FUNCTION_BLOCK Valvula_Saida_Digital_HMI (* Service Interface Function Block Type *)
  (* Standard: 61499-2 *)
  (* Version 0.0, 1/26/2026, Schneider Electric, template *)
  PACKAGE Hidryco.HidrycoLib;
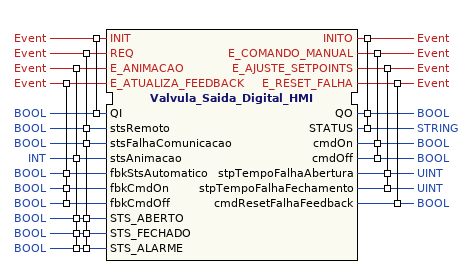
  EVENT_INPUT
    INIT WITH QI;
    REQ WITH stsRemoto, stsFalhaComunicacao, STS_ABERTO, STS_FECHADO, STS_ALARME;
    E_ANIMACAO WITH stsAnimacao, STS_ABERTO, STS_FECHADO, STS_ALARME;
    E_ATUALIZA_FEEDBACK WITH fbkStsAutomatico, fbkCmdOn, fbkCmdOff;
  END_EVENT
  EVENT_OUTPUT
    INITO WITH QO, STATUS;
    E_COMANDO_MANUAL WITH cmdOn, cmdOff;
    E_AJUSTE_SETPOINTS WITH stpTempoFalhaAbertura, stpTempoFalhaFechamento;
    E_RESET_FALHA WITH cmdResetFalhaFeedback;
  END_EVENT
  VAR_INPUT
    QI : BOOL;
    stsRemoto : BOOL;
    stsFalhaComunicacao : BOOL;
    stsAnimacao : INT;
    fbkStsAutomatico : BOOL;
    fbkCmdOn : BOOL;
    fbkCmdOff : BOOL;
    STS_ABERTO : BOOL;
    STS_FECHADO : BOOL;
    STS_ALARME : BOOL;
  END_VAR
  VAR_OUTPUT
    QO : BOOL; (* Event Output Qualifier *)
    STATUS : STRING; (* Service Status *)
    cmdOn : BOOL;
    cmdOff : BOOL;
    stpTempoFalhaAbertura : UINT;
    stpTempoFalhaFechamento : UINT;
    cmdResetFalhaFeedback : BOOL;
  END_VAR
  SERVICE /
    SEQUENCE 
    END_SEQUENCE
  END_SERVICE
END_FUNCTION_BLOCK
